Omron CX-Programmer project Karosszeria_gyartosor (CX-Programmer 9.10)

# PLC PLC: CJ2M CPU32
I/O table (CPU CJ2M-CPU32): rack 0 slot 11 CJ2M-EIP21

## Global symbols (name address type ; comment)
Cell_1_Speed D0.05 BOOL  ; Az első cellában beállítható sebesség.
Cell_2_Speed D0.04 BOOL  ; A második cellában beállítható sebesség.
Global_START D0.06 BOOL  ; A robotpozíciók érvényesítő bitjének állapota.
Global_STOP D0.03 BOOL  ; A vészstop jelzőbitje.
INPUT 2 UINT  ; A vezérlés bemenete.
IN_Acknowledgement 2.13 BOOL  ; Nyugtázás
IN_Body_Type_B0 2.00 BOOL  ; Utoljára beadott karosszéria típusa
IN_Body_Type_B1 2.01 BOOL  ; Utoljára beadott karosszéria típusa
IN_Emergency_Stop 2.14 BOOL  ; Vészstop
IN_Operator_Movement 2.08 BOOL  ; Operátor mozgása
IN_Robot_1_Done 2.09 BOOL  ; Robot 1 mozgás befejezve
IN_Robot_2_Done 2.10 BOOL  ; Robot 2 mozgás befejezve
IN_Robot_3_Done 2.11 BOOL  ; Festőrobot mozgás befejezve
IN_Sensor_Cell_1 2.05 BOOL  ; Cella 1
IN_Sensor_Cell_1_Arrival 2.02 BOOL  ; Cella 1 érkezés
IN_Sensor_Cell_2 2.06 BOOL  ; Cella 2
IN_Sensor_Cell_2_Arrival 2.03 BOOL  ; Cella 2 érkezés
IN_Sensor_Cell_3 2.07 BOOL  ; Cella 3
IN_Sensor_Cell_3_Arrival 2.04 BOOL  ; Cella 3 érkezés
IN_Unused 2.15 BOOL  ; Nincs használatban
IN_Warm_Reset 2.12 BOOL  ; Factory reset (warm reset)
OUTPUT 3 UINT  ; A vezérlés kimenete.
OUT_Belt_1_Switch 3.09 BOOL  ; Futószalag 1
OUT_Belt_2_Switch 3.10 BOOL  ; Futószalag 2
OUT_Belt_3_Switch 3.11 BOOL  ; Futószalag 3
OUT_Crane_Effector 3.15 BOOL  ; Daru megfogó vezérlése
OUT_Crane_Position_B0 3.12 BOOL  ; Daru pozíció
OUT_Crane_Position_B1 3.13 BOOL  ; Daru pozíció
OUT_Crane_Position_B2 3.14 BOOL  ; Daru pozíció
OUT_Robot_Effector 3.07 BOOL  ; Hegesztőpisztoly vagy a festékszóró vezérlése
OUT_Robot_Position_B0 3.04 BOOL  ; Robot adott konfiguráció vezérlése
OUT_Robot_Position_B1 3.05 BOOL  ; Robot adott konfiguráció vezérlése
OUT_Robot_Position_B2 3.06 BOOL  ; Robot adott konfiguráció vezérlése
OUT_Robot_Select_B0 3.00 BOOL  ; Robot kiválasztása
OUT_Robot_Select_B1 3.01 BOOL  ; Robot kiválasztása
OUT_Robot_Speed 3.02 BOOL  ; Robot lassú-gyors
OUT_Robot_Start 3.08 BOOL  ; Robotmozgás érvényesítés
OUT_Robot_Stop 3.03 BOOL  ; Robot állj
Operation_Sequence_1 D5 UINT[11]  ; Az 1-es típusú karosszérián elvégezendő hegesztési munkálatok pozícióit tartalmazó tömb.
Operation_Sequence_2 D19 UINT[11]  ; Az 2-es és 3-as típusú karosszériákon elvégezendő hegesztési munkálatok pozícióit tartalmazó tömb.
Operation_Sequence_3 D41 UINT[6]  ; A karosszériákon elvégezendő festési munkálatok pozícióit tartalmazó tömb.

## Program NewProgram1 (cyclic task 0)
Local symbols
BIN_Array W10.00 BOOL[16]
UINT_Value W10 UINT

### Section Section1

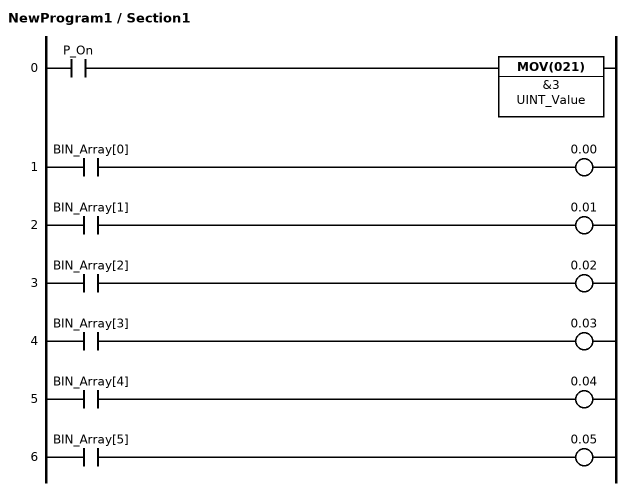
; rung 0
LD P_On
MOV(021) &3 UINT_Value
; rung 1
LD BIN_Array[0]
OUT 0.00
; rung 2
LD BIN_Array[1]
OUT 0.01
; rung 3
LD BIN_Array[2]
OUT 0.02
; rung 4
LD BIN_Array[3]
OUT 0.03
; rung 5
LD BIN_Array[4]
OUT 0.04
; rung 6
LD BIN_Array[5]
OUT 0.05

### Section END
; rung 0
END(001)